// Mitsubishi GX Works2 project: mov연습   PLC: Q02/Q02H

PROGRAM MAIN
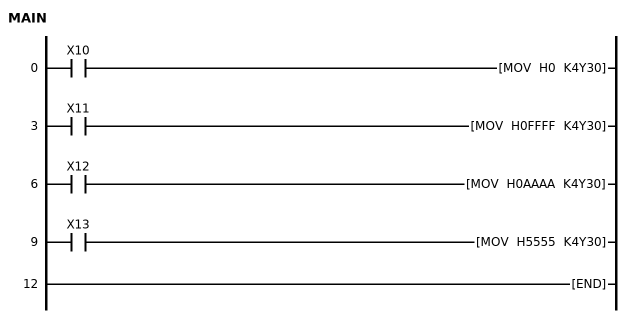
0     LD      X10
      MOV     H0 K4Y30
3     LD      X11
      MOV     H0FFFF K4Y30
6     LD      X12
      MOV     H0AAAA K4Y30
9     LD      X13
      MOV     H5555 K4Y30
12    END
END_PROGRAM
